FUNCTION f_BitDel : T_PROCESS
VAR_INPUT
  inVal   : T_PROCESS;
  bitNo   : DINT;
END_VAR
VAR
  wConst : T_PROCESS := 1;
END_VAR

IF ( inVal AND SHL( wConst,TO_SINT(bitNo) MOD TO_INT(SIZEOF(T_PROCESS)*8) ) ) > 0 THEN
  f_BitDel := inVal XOR (SHL( wConst,TO_SINT(bitNo) MOD TO_INT(SIZEOF(T_PROCESS)*8) ));
ELSE
  f_BitDel := inVal;
END_IF

END_FUNCTION

(* stored: Version 1.1.0.1
   POU f_BitDel: Id {6417603d-b229-4ca2-bc92-1faa058378c2}, SpecialFunc None *)
